FUNCTION_BLOCK T_GripperManualMode EXTENDS T_NamedBase IMPLEMENTS I_PackMode
VAR
	_gripper : I_GripperModule;
END_VAR

METHOD Initialise
VAR_INPUT
	Gripper : I_GripperModule;
END_VAR
_gripper := Gripper;
END_METHOD

END_FUNCTION_BLOCK

(* stored: Version 1.1.0.1, ProductVersion 3.1.4024.12
   POU T_GripperManualMode: Id {77faa915-6ddf-4717-8420-89f4dde5a135}, SpecialFunc None
   Method Initialise: Id {2026c3b5-73a5-47a5-92b0-1284bcfe0625} *)
